{attribute addProperty BoxType "AT2000-0233-0022"}
{attribute addProperty Id "StatusAT %I*UINT1621Current_actual_value_ChAT %I*ARRAY[0 ..13] OF INT224280"}
{attribute addProperty CRC "987499732"}
{attribute addProperty SizeInBites "240"}
{attribute addProperty SizeInBytes "30"}
TYPE CC_Inputs_14_Ch_5FB71CBE :
STRUCT
	{attribute addProperty Name "Status"}
	Status AT %I* : UINT;
	{attribute addProperty Name "Current_actual_value_Ch"}
	Current_actual_value_Ch AT %I* : ARRAY[0 ..13] OF INT;
END_STRUCT
END_TYPE

(* stored: Version 1.2.0.0, ProductVersion 3.1.4024.9
   DUT CC_Inputs_14_Ch_5FB71CBE: Id {081d1af9-589d-4aaf-8a4c-27950d281da3} *)
